Staubli VAL3: goToPoint.pgx

public program goToPoint(num x_nIndexGun)
begin
  resetMotion()
  if x_nIndexGun==0
    movej(saveTool:rif2,saveTool:gun[x_nIndexGun],{25,25,25,9999,9999,off,50,50})
  else
    pPoint.trsf=position(saveTool:rif2,world)
    pPoint.config={sfree,efree,wfree}
    movej(pPoint,saveTool:gun[x_nIndexGun],{25,25,25,9999,9999,off,50,50})
  endIf
end
